# EPICS substitutions: ek9000App/Db/userHost.substitutions
# Example substitutions file

file "db/dbExample1.db" {
    { user = "jeremyHost" }
}

file db/dbExample2.db {
    pattern { user, no, scan }
        { "jeremyHost", 1, "1 second" }
        { "jeremyHost", 2, "2 second" }
        { "jeremyHost", 3, "5 second" }
}
